PROGRAM Prg_FSM
VAR
	Start: BOOL;
	Stop: BOOL;
	Mixer: BOOL;
	Pump: BOOL;
	Gate: BOOL;
	Timer1: TON;
	State: INT;
	StartT: R_TRIG;
	StopT: R_TRIG;
END_VAR


StartT(CLK:=Start);
StopT(CLK:=Stop);

CASE State OF
	0:
		IF StartT.Q THEN
			State:=1;
		ELSE
			State:=0;
		END_IF
	
	1:
		Mixer:=TRUE;
		Timer1(IN:=TRUE, PT:=T#5S, ET=>);
		IF Timer1.Q THEN
			Timer1(IN:=FALSE);
			State:=2;
		END_IF
	2:
		Pump:=TRUE;
		Timer1(IN:=TRUE, PT:=T#5S, ET=>);
		IF Timer1.Q THEN
			Timer1(IN:=FALSE);
			pump:=FALSE;
			State:=3;
		ELSE
			State:=2;
		END_IF
	3:
		Timer1(IN:=TRUE, PT:=T#5S, ET=>);
		IF Timer1.Q THEN
			Timer1(IN:=FALSE);
			Mixer:=FALSE;
			State:=4;
		ELSE
			State:=3;
		END_IF
	4:
		Gate:=TRUE;
		Timer1(IN:=TRUE, PT:=T#5S, ET=>);
		IF Timer1.Q THEN
			Timer1(IN:=FALSE);
			Gate:=FALSE;
			state:=0;
		ELSE
			State:=4;			
		END_IF
	
END_CASE

IF StopT.Q THEN
	State:=0;
	Mixer:=FALSE;
	Pump:=FALSE;
	Gate:=FALSE;
END_IF

END_PROGRAM

(* stored: Version 1.1.0.1, ProductVersion 3.1.4024.9
   POU Prg_FSM: Id {f8af83b1-368f-46d9-a817-42c4bb083253}, SpecialFunc None *)
